Staubli VAL3: generation_generator.pgx

program generation_generator(num x_nDays)
  local num l_nElement
  local num l_nValue
  local num l_nDays
  local num l_nNewFishes
  local num l_nRESULT
begin

  // count values
  resize(nCounter,1,1)
  nCounter = 0
  resize(nCounter,1,9)
  for l_nElement = 0 to size(nInput)-1
    for l_nValue = 0 to 8
      if nInput[l_nElement] == l_nValue
        nCounter[l_nValue] = nCounter[l_nValue] + 1
      endIf
    endFor
  endFor

  for l_nDays = 1 to x_nDays
    l_nNewFishes = nCounter[0]

    delete(nCounter[0])

    nCounter[6] = nCounter[6] + l_nNewFishes
    append(nCounter)
    nCounter[8] = l_nNewFishes
  endFor

  call math:sum(nCounter, l_nRESULT)
  call util:printNum(l_nRESULT)


end
